FUNCTION_BLOCK RobotA22 EXTENDS KukaRobot
VAR_INPUT
	wrapSafety AT %Q* : BOOL;
END_VAR
VAR_OUTPUT //from outputs array
	taskID AT %Q* : TaskA22;
	param1 AT %Q* : INT;
	param2 AT %Q* : INT;
	Xmm AT %Q* : INT;
	Ymm AT %Q* : INT;
	Zmm AT %Q* : INT;
	angle AT %Q* : INT;
	foldPosition0 AT %Q* : INT;
	foldPosition1 AT %Q* : INT;
END_VAR
VAR_OUTPUT //from inputs array
	tool : SectionEnum := SectionEnum.CARDBOARD_CORNERGUARD;
	suspendedMaterial : STRING;
	
	completedTask AT %I* : TaskA22;
	eoatDistance AT %I* : INT;
	cardboardAvailability AT %I* : INT;
	cornerGuardAvailability AT %I* : INT;
	materialAtHoldingPosition AT %I* : INT;
	//grp6	
	wrapSafetyIn AT %I* : BOOL;
END_VAR
VAR //HMI data
	reservationEnum : SectionEnum;
	hmiTask : STRING;
	hmiTool : STRING;
END_VAR

{warning disable C0195}

SUPER^();

reservationEnum := reservation;
IF reservationEnum = SectionEnum.NULL_SECTION THEN
	hmiReservation := 'N/A';
ELSE
	hmiReservation := TO_STRING(reservationEnum);
END_IF

hmiTask := TO_STRING(taskID);
hmiTool := TO_STRING(tool);

{attribute 'monitoring' := 'call'}
PROPERTY Busy : BOOL
GET
VAR
	//emptyOutput : ARRAY[1..50] OF INT;
END_VAR
//Busy stays TRUE until outputs are cleared AND completed task has elapsed
//Ready is always inverse of Busy
Busy := taskID <> 0 OR completedTask <> 0;
END_GET
END_PROPERTY

METHOD changeEOAT : BOOL
VAR_INPUT
	targetTool : SectionEnum;
END_VAR
//fill in IO here

changeEOAT := TRUE;
END_METHOD

METHOD clearCommand : BOOL
VAR_INPUT
END_VAR
taskID := 0;
param1 := 0;
param2 := 0;
Xmm := 0;
Ymm := 0;
Zmm := 0;
angle := 0;
foldPosition0 := 0;
foldPosition1 := 0;
END_METHOD

{attribute 'monitoring' := 'call'}
PROPERTY Done : BOOL
GET
Done :=
	completedTask = taskID AND
	taskID <> 0 AND
	completedTask <> 0;
END_GET
END_PROPERTY

{attribute 'monitoring' := 'call'}
PROPERTY HoldMaterial : STRING
GET
HoldMaterial := suspendedMaterial;
END_GET
SET
suspendedMaterial := HoldMaterial;
END_SET
END_PROPERTY

{attribute 'monitoring' := 'call'}
PROPERTY Ready : BOOL
GET
Ready := taskID = 0 AND completedTask = 0;
END_GET
END_PROPERTY

METHOD setParameters : BOOL
VAR_INPUT
	newTaskID : INT;
	newParam1 : INT;
	newParam2 : INT;
	newXmm : INT;
	newYmm : INT;
	newZmm : INT;
	newAngle : INT;
	newFoldPos0 : INT;
	newFoldPos1 : INT;
END_VAR
VAR_INPUT
	newWrapSafety : BOOL;
END_VAR
taskID := newTaskID;
param1 := newParam1;
param2 := newParam2;
Xmm := newXmm;
Ymm := newYmm;
Zmm := newZmm;
angle := newAngle;
foldPosition0 := newFoldPos0;
foldPosition1 := newFoldPos1;

wrapSafety := newWrapSafety;
END_METHOD

END_FUNCTION_BLOCK

(* stored: Version 1.1.0.1, ProductVersion 3.1.4024.11
   POU RobotA22: Id {154e6fc8-e169-4c7b-8aba-d1a085cf4a2c}, SpecialFunc None
   Folder Properties: Id {0b1bba9e-3c27-4acf-96f1-477bb38b27ac}
   Property Busy: Id {47b197a8-c1d1-47ef-a3bf-548c3d5538e8}
   Get Get: Id {e58a7940-91e9-487f-8510-ef610e80aaee}
   Method changeEOAT: Id {91eaa1e0-fe94-4b42-a50f-6867ae73bcb6}
   Method clearCommand: Id {81d6ba48-6744-4d4c-9e10-3eb71ebc4f31}
   Property Done: Id {011f33cf-69d3-4e4f-aa25-727436880bee}
   Get Get: Id {033291ab-ebbd-4a21-b480-92e50b83ef3e}
   Property HoldMaterial: Id {00ac4986-a380-421e-8575-2cbfef1d8f83}
   Get Get: Id {55579013-334a-4608-b4ed-ed7f0eaba012}
   Set Set: Id {2e53f269-18e0-4d5f-8ac4-9085b32a35c1}
   Property Ready: Id {b20cbaf9-6ae2-4067-9bd9-40dbc5c522b9}
   Get Get: Id {13684114-f5cb-4dd5-9172-eaceacf67fb8}
   Method setParameters: Id {200a31c1-2c60-45e5-bfd7-a4fcac794d1b} *)
